PROGRAM MAIN
VAR
END_VAR

master.dummyAction();
slave.dummyAction();

couple.checkGearIn();
couple.checkGearOut();

master.checkPower();
slave.checkPower();

master.checkSetPoint();
slave.checkSetPoint();


master.checkMoving();
master.checkRelMove();

master.checkReset();
master.checkStop();
master.checkGoHome();

END_PROGRAM

(* stored: Version 1.1.0.1, ProductVersion 3.1.4024.4
   POU MAIN: Id {4ca54771-8ae5-4549-901f-6cb523f28aef}, SpecialFunc None *)
